// TIA Portal V20 export
DATA_BLOCK "InstSleepModeManager"   // DB293
// stored: InstanceOfName LER_SleepModeManager, InstanceOfType FB
"LER_SleepModeManager"
   // VAR_INPUT
   //    enable : Bool;
   //    unitStatus : "LAF_typeUnitStatus";
   //    wakeUpReq : Bool;
   //    sleepDelay : Time;
   //    deepSleepDelay : Time;
   // END_VAR
   // VAR_OUTPUT
   //    sleepModeChangeReq : Bool;
   //    deepSleepModeChangeReq : Bool;
   //    wakeUpRecoveryRequired : Bool;
   // END_VAR
   // VAR
   //    instSleepDelay { ExternalAccessible := 'False'; ExternalVisible := 'False'; ExternalWritable := 'False'; S7_SetPoint := 'True'} : TON_TIME;
   //    instDeepSleepDelay { ExternalAccessible := 'False'; ExternalVisible := 'False'; ExternalWritable := 'False'; S7_SetPoint := 'True'} : TON_TIME;
   //    statStandbyReady { ExternalAccessible := 'False'; ExternalVisible := 'False'; ExternalWritable := 'False'} : Bool;
   //    statWakeUpRecoveryRequired { ExternalAccessible := 'False'; ExternalVisible := 'False'; ExternalWritable := 'False'} : Bool;
   // END_VAR
BEGIN
END_DATA_BLOCK
